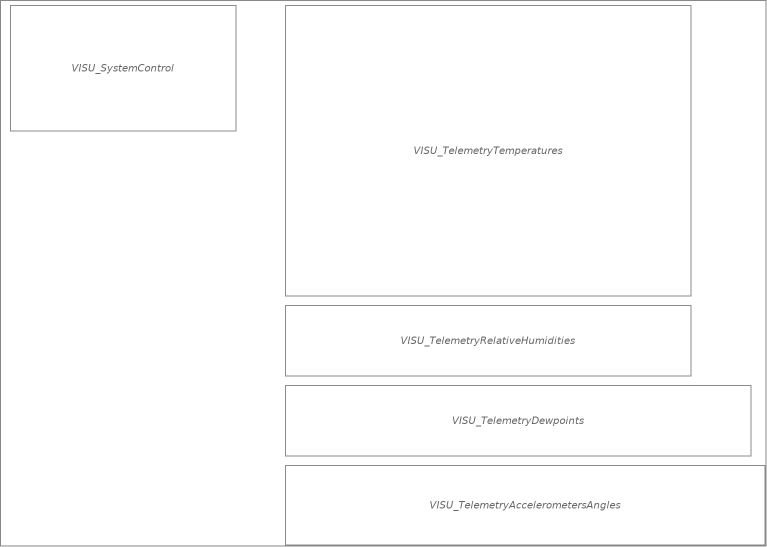
VISUALIZATION VISU_TelemetryOverview  // 767x547
VAR_IN_OUT
	ref : Telemetry;
    widget : TelemetryWidget;
END_VAR
    Frame (10,5 226x126)
        shows VISU_SystemControl(status := widget.actualStatus, button_initialize := widget.button_initialize, button_operating := widget.button_operating, button_locking := widget.button_locking)
    Frame (285,5 406x291)
        shows VISU_TelemetryTemperatures(ref := ref.parts.temperatures, widget := widget.temperatures)
    Frame (285,305 406x71)
        shows VISU_TelemetryRelativeHumidities(ref := ref.parts.relativeHumidities, widget := widget.relativeHumidities)
    Frame (285,385 466x71)
        shows VISU_TelemetryDewpoints(ref := ref.parts.dewpoints, widget := widget.dewpoints)
    Frame (285,465 480x80)
        shows VISU_TelemetryAccelerometersAngles(ref := ref.parts.accelerometers, widget := widget.accelerometers)
END_VISUALIZATION

(* stored: Version 1.1.0.1, ProductVersion 3.1.4019.2
   Visu VISU_TelemetryOverview: Id {ef4e4c95-2490-4cfd-a4e0-70aaab02477e} *)
